TYPE ST_MetaData :
STRUCT
  BatteryVoltage : DINT;
  VoltageUnit : STRING;
  ClickType : STRING;
  SensorValue1 : DINT;
END_STRUCT
END_TYPE

(* stored: Version 1.1.0.1, ProductVersion 3.1.4024.12
   DUT ST_MetaData: Id {fc33f874-ae3b-48cc-be60-d9235c23eecf} *)
